// TwinCAT 3 PLC project PLC
// ProgramVersion: 3.1.4026.19
// CompilerDefines: VISU_USEPROPERTYINFO
// libraries:
//   Tc2_Standard, * (Beckhoff Automation GmbH)
//   Tc2_System, * (Beckhoff Automation GmbH)
//   VisuSymbols, 4.5.0.0 (System)
// project tree:
//   / GlobalTextList.TcGTLO, PlcTask.TcTTO, Visualization Manager.TcVMO (not stored)
//   POUs/ MAIN.TcPOU
//   VISUs/ Visualization.TcVIS
// real-time tasks:
//   TASK PlcTask: cycle T#10ms, priority 20, ADS port 350

CONFIGURATION PLC
    RESOURCE PLC ON TwinCAT3
        TASK PlcTask(INTERVAL := T#10ms, PRIORITY := 20);
        PROGRAM MAIN WITH PlcTask : MAIN;
    END_RESOURCE
END_CONFIGURATION

// ---- POUs/MAIN.TcPOU
PROGRAM MAIN
VAR
    bButton : BOOL;   // Buton (giris) - simdilik sanal
    bLED    : BOOL;   // LED (cikis)  - simdilik sanal
END_VAR

bLED := bButton;

END_PROGRAM

// ---- GlobalTextList.TcGTLO
TEXTLIST GlobalTextList
  586 = 'Button'
END_TEXTLIST

// ---- VISUs/Visualization.TcVIS
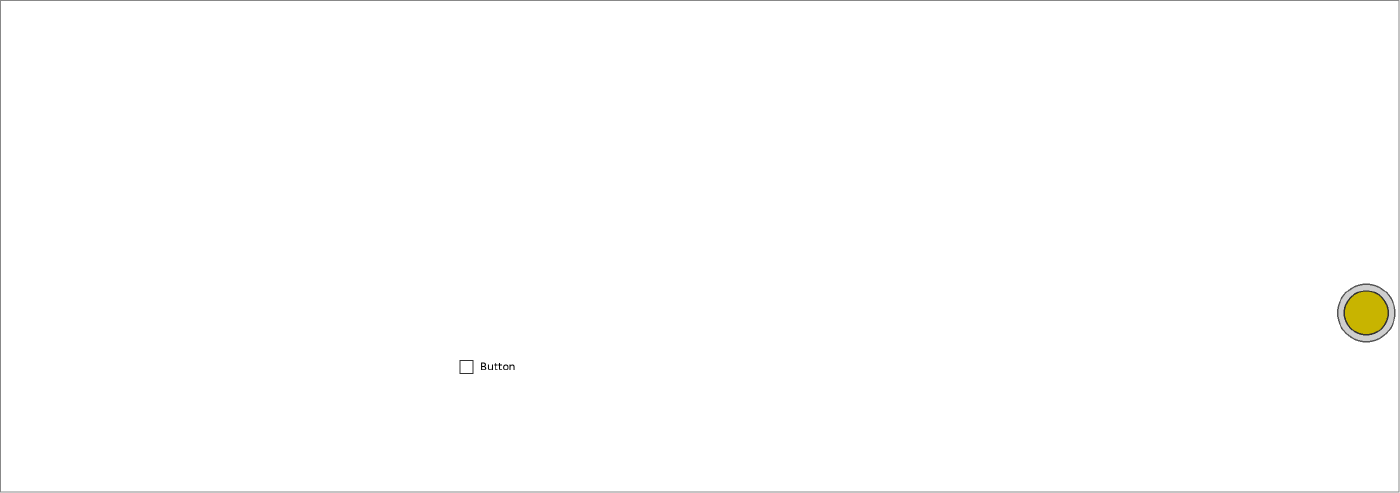
VISUALIZATION Visualization  // 1453x512
    Checkbox (475,250 326x262), "Button", variable: MAIN.bButton
    Lamp1 (1383,290 70x70), variable: MAIN.bLED, style: Lamp-Lamp1-Yellow
END_VISUALIZATION
